(* Zaleca się ustawienie tolerancji na poziomie 3%. lrOffsetPercentValue := 3*)

FUNCTION_BLOCK FB_BalluffBMP0005
VAR_INPUT
	diSensorMeasurementValue	AT%I*		: DINT;						//IOLink zmienna z czujnika balluff
	lrOffsetPercentValue					: LREAL;					//To jest tolerancja Otwarcia/Zamknięcia (Podajesz w procentach od 1-100 %)
	
	bRecipeChanged							: BOOL;						//Receptura została zmieniona 
	//Kalibracja
	bCalibration							: BOOL;						//Czujnika wymaga kalibracji, żeby przejść w tryb kalibracji musicie bCalibration wystawić na TRUE
	bAcceptOpenCalibrationValue				: BOOL;						//Procedura kalibracji, Operator potwierdza że chwytak jest otwarty. Przepisuję wartość iolink do zmiennej local
	bAcceptCloseCalibrationValue			: BOOL;						//Procedura kalibracji, Operator potwierdza że chwytak złapał butelkę. Przepisuję wartość iolink do zmiennej local.
	
	sStationName							: STRING(200);
	
END_VAR
VAR_OUTPUT
	bSensorClose							: BOOL;						//Wystawia true, gdy chwytak jest otwarty a wartość czujnika iolink mieści się w zakresie tolerancji 
	bSensorOpen								: BOOL;						//Wystawia true, gdy chwytak jest zamknięty a wartość czujnika mieści się w zakresie tolerancji
	bWarning								: BOOL;						//Ostrzeżenie
	sWarningDescription						: STRING(200);				//Opis ostrzeżenia
	sSensorName								: STRING(200);
	iCalibrationState						: INT;						//Aktualny krok kalibracji
	bCalibrationDone						: BOOL;						// Potwierdzenie popranej kalibracji czujnika
END_VAR
VAR
	tonOpenSensor							: TON;
	tonCloseSensor							: TON;
	
	rtRecipeChanged							: R_TRIG;
	rtCalibration							: R_TRIG;
	
	
	lrCalibrationOpenValue					: LREAL;
	lrCalibrationCloseValue					: LREAL;
	bOpen									: BOOL;
	bClose									: BOOL;
END_VAR

ACT_Warnings();
ACT_Calibration();
ACT_Signals();

ACTION ACT_Calibration:
rtCalibration(CLK:= bCalibration);
rtRecipeChanged(CLK:= bRecipeChanged);


IF rtRecipeChanged.Q THEN
	bCalibrationDone				:= FALSE;
	lrCalibrationOpenValue			:= 0;
	lrCalibrationCloseValue			:= 0;
END_IF

IF rtCalibration.Q AND iCalibrationState <> 0 THEN
	bCalibrationDone				:= FALSE;
	lrCalibrationOpenValue			:= 0;
	lrCalibrationCloseValue			:= 0;
	iCalibrationState				:= 10;
END_IF

CASE iCalibrationState OF
	
	0:
		IF rtCalibration.Q THEN
			bCalibrationDone		:= FALSE;
			lrCalibrationOpenValue	:= 0;
			lrCalibrationCloseValue	:= 0;
			iCalibrationState		:= 10;
		END_IF
		
	10:
		IF bAcceptOpenCalibrationValue THEN
			
			lrCalibrationOpenValue	:= diSensorMeasurementValue;
			iCalibrationState		:= 20;
		END_IF
		
	20:
		IF bAcceptCloseCalibrationValue THEN
			
			bCalibrationDone		:= TRUE;
			
			lrCalibrationCloseValue	:= diSensorMeasurementValue;
			iCalibrationState		:= 0;
		END_IF
		
		
END_CASE
END_ACTION

ACTION ACT_Signals:
tonOpenSensor(IN:= bOpen, PT:= T#50MS);
tonCloseSensor(IN:= bClose, PT:=  T#50MS);

IF lrOffsetPercentValue = 0 THEN	
	lrOffsetPercentValue		:= 1;	
END_IF

IF bCalibrationDone THEN

	IF (diSensorMeasurementValue <= lrCalibrationOpenValue + 10000)(*(lrCalibrationOpenValue* (lrOffsetPercentValue/100)))*) AND
	   (diSensorMeasurementValue >= lrCalibrationOpenValue - 10000)(*(lrCalibrationOpenValue* (lrOffsetPercentValue/100)))*) THEN
	
		bOpen					:= TRUE;	   
	   	bSensorOpen				:= tonOpenSensor.Q;//TRUE;
	   
	ELSE
		
		bOpen					:= FALSE;
		bSensorOpen				:= FALSE;
	END_IF
	
	
	
	
	IF ((diSensorMeasurementValue <= lrCalibrationCloseValue + lrOffsetPercentValue)(*(lrCalibrationCloseValue* (lrOffsetPercentValue/100)))*) AND
	   (diSensorMeasurementValue >= lrCalibrationCloseValue - lrOffsetPercentValue)(*(lrCalibrationCloseValue* (lrOffsetPercentValue/100)))*) )OR
		(diSensorMeasurementValue <= - 4692 + 200 AND diSensorMeasurementValue >=  - 4692 - 200) THEN
		
		bClose					:= TRUE;   
	   	bSensorClose			:= tonCloseSensor.Q;//TRUE;
	   
	ELSE
		bClose					:= FALSE;
		bSensorClose			:= FALSE;	
	END_IF

ELSE
	
	bSensorOpen					:= FALSE;
	bSensorClose				:= FALSE;
END_IF
END_ACTION

ACTION ACT_Warnings:

IF NOT bCalibrationDone AND NOT bWarning THEN
	
	bWarning				:= TRUE;
	sWarningDescription		:= 'Czujnik wymaga kalibracji';
	sSensorName				:= sStationName;
END_IF

//Reset warningów
IF bCalibrationDone THEN
	bWarning				:= FALSE;
	sWarningDescription		:= '';
	sSensorName				:= '';
END_IF
END_ACTION

END_FUNCTION_BLOCK

(* stored: Version 1.1.0.1, ProductVersion 3.1.4026.13, FileIdentifier 21dac51c531bbf7c9023c2ff8a067f1bc71359ff, FileSignature 5553cddfb0ef073d5909a72a2fea14fd52f5214ff0536fbff3f96da7cff26623ad7cf664be4ca638c6bf580351e929ec658efd871b5c5907d2a2a58cc3c95a2b7b036c86118fc10a6e3c88937282b8816a2794888ae8d69c8e470dbd7e44f9ff8b46ed4c0f13786495fe27401b80a55556952477648ece22c065c4764b6d09907dd42c30c5d2fbfc141428eb2d969992b76dcf225f67159fb7fe293ef4ea2c60b789d84e5f350b2365a3249fa6acd8663b653c12fd25b3cfe3cc18d91739b4d51924829331e4b17668758f60231c0bd20bef4550d9d0aecf65386c544ca2ffaa481c091e4ca2c4e8cec6beabc8b5c3c6482207f9775ff1cf08d5c181eac603b6
   POU FB_BalluffBMP0005: Id {8d3a5723-7faa-4c83-af28-bc7423195b78}, SpecialFunc None
   Action ACT_Calibration: Id {d98b9fa4-586a-4cee-995b-6d10c1a394ce}
   Action ACT_Signals: Id {2e7719e6-2c18-4fb9-9e53-f13548269a02}
   Action ACT_Warnings: Id {e9cb5a09-0d80-471b-a62d-b4d1432ab632} *)
